Staubli VAL3: RobotStatusMsg.dtx

public Body body
  [0]
    num nData[32]
public Header header
  [0]
    num nMsgType
    num nCommType
    num nReplyCode
    num nData[12]
public Prefix prefix
  [0]
    num nLength
    num nData[4]
public RobotStatus robotStatus
  [0]
    num nDrivesPowered
    num nEStopped
    num nErrorCode
    num nInError
    num nInMotion
    num nMode
    num nMotionPossible
    num nTrajComplete
